FUNCTION_BLOCK IAS_Skill_MUX (* Composite Function Block Type *)
  (* Standard: 61499-2 *)
  (* Version 1.0, 2019-07-03, dorofeev *)
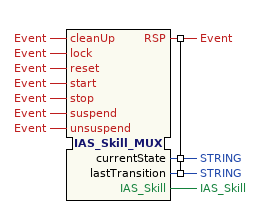
  EVENT_INPUT
    cleanUp; (* Initialization Request *)
    lock; (* Normal Execution Request *)
    reset;
    start;
    stop;
    suspend;
    unsuspend;
  END_EVENT
  EVENT_OUTPUT
    RSP WITH currentState, lastTransition;
  END_EVENT
  VAR_OUTPUT
    currentState : STRING;
    lastTransition : STRING;
  END_VAR
  PLUGS
    IAS_Skill : IAS_Skill;
  END_PLUGS
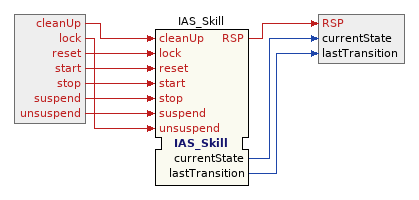
  EVENT_CONNECTIONS
    cleanUp TO IAS_Skill.cleanUp;
    lock TO IAS_Skill.lock;
    reset TO IAS_Skill.reset;
    start TO IAS_Skill.start;
    stop TO IAS_Skill.stop;
    suspend TO IAS_Skill.suspend;
    unsuspend TO IAS_Skill.unsuspend;
    IAS_Skill.RSP TO RSP;
  END_CONNECTIONS
  DATA_CONNECTIONS
    IAS_Skill.currentState TO currentState;
    IAS_Skill.lastTransition TO lastTransition;
  END_CONNECTIONS
END_FUNCTION_BLOCK
